PROGRAM Alarms
VAR
	Alarms_Array : ARRAY [0..255] OF BOOL; //this is the alarms array for all the alarms of a given system. if a larger arry in needed eiter use to Bit Counter functions or change FOR loop in Bit Counter to much bigger array.
	Temp_AlarmCnt : UINT;
	AlarmCnt : UINT; //number of active alarms
	AlarmExist : BOOL; //ON as long as there is an active alarm
	Alarm_SR : SR; //SR replace KEEP in Omron progrem for Alarm Relay
	Alarm_Relay AT%Q* : BOOL; //Alarm Relay R10
END_VAR
VAR // added by the converter: edge detectors and wires of the graphical bodies
    _w1, _w2, _w3 : BOOL;
END_VAR

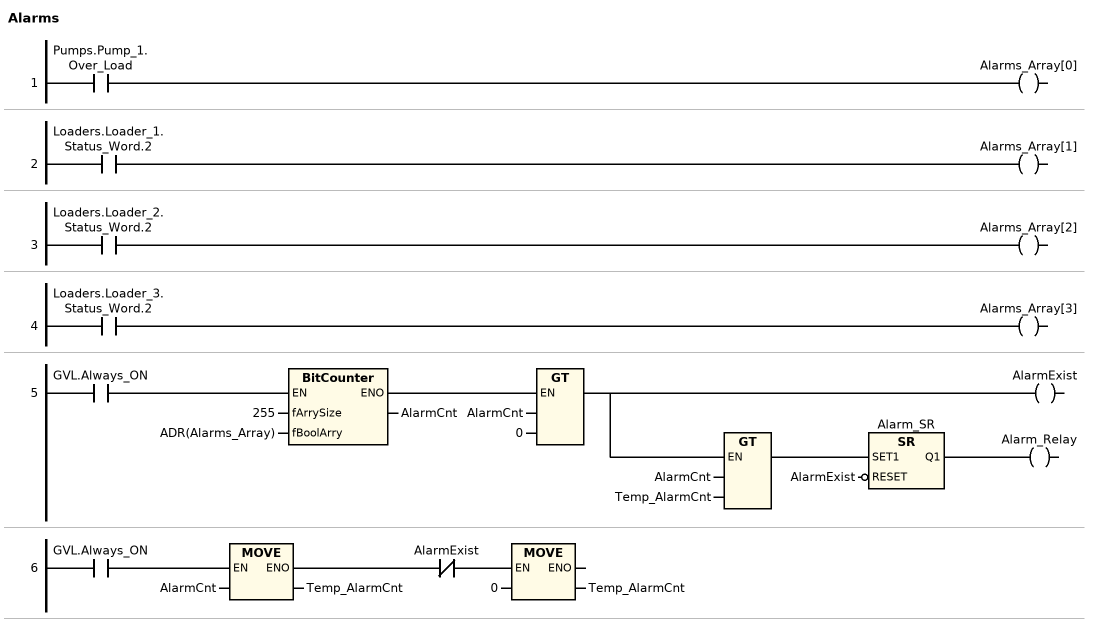
// NETWORK 1
Alarms_Array[0] := Pumps.Pump_1.Over_Load;

// NETWORK 2
Alarms_Array[1] := Loaders.Loader_1.Status_Word.2;

// NETWORK 3
Alarms_Array[2] := Loaders.Loader_2.Status_Word.2;

// NETWORK 4
Alarms_Array[3] := Loaders.Loader_3.Status_Word.2;

// NETWORK 5
_w1 := GVL.Always_ON;
IF _w1 THEN AlarmCnt := BitCounter(fArrySize := 255, fBoolArry := ADR(Alarms_Array)); END_IF
_w2 := _w1 AND AlarmCnt > 0;
AlarmExist := _w2;
Alarm_SR(SET1 := _w2 AND AlarmCnt > Temp_AlarmCnt, RESET := NOT AlarmExist); // SR
Alarm_Relay := Alarm_SR.Q1;

// NETWORK 6
_w3 := GVL.Always_ON;
IF _w3 THEN Temp_AlarmCnt := AlarmCnt; END_IF
IF _w3 AND NOT AlarmExist THEN Temp_AlarmCnt := 0; END_IF

END_PROGRAM

(* stored: Version 1.1.0.1, ProductVersion 3.1.4024.13
   POU Alarms: Id {e4fd9ffa-2814-4d15-85d2-737d9e46af6b}, SpecialFunc None *)
